PROGRAM MAIN
VAR

    fbLogHandler : FB_LogHandler;
    i:INT;
END_VAR

i := i + 1;

fbLogHandler();

(* FEE devices*)
PRG_FEE();
PRG_PMPS();
PRG_FSV_Interfaces();

(*  *)

(*Hutch*)
PRG_Hutch_Gauges();
PRG_Hutch_Beamline_Valves();
PRG_Roughing_Pumps();
PRG_Hutch_Ion_Pumps();

PRG_IP1_ECAT_Interfaces();
PRG_HV_SAFETY();

END_PROGRAM

(* stored: Version 1.1.0.1, ProductVersion 3.1.4022.18
   POU MAIN: Id {53e436ba-9af9-4ca4-ad7b-a6b2399fa417}, SpecialFunc None *)
